{attribute 'qualified_only'}
{attribute 'strict'}
TYPE E_CAN_Object_Test_Error_Bits :
(
	No_error := 0
	
) WORD;
END_TYPE

(* stored: Version 1.1.0.1, ProductVersion 3.1.4024.11
   DUT E_CAN_Object_Test_Error_Bits: Id {d313b95c-6e46-490a-8863-b138b30eb387} *)
